{attribute 'qualified_only'}
VAR_GLOBAL
	iInput AT%I* : INT;
END_VAR

(* stored: Version 1.1.0.1, ProductVersion 3.1.4024.12
   GVL GVL_IO: Id {3fc50ee0-781f-485a-9f08-dd256e844bfc} *)
